(* CoDeSys 2.3 export: GVL_SYMBOLSANDDATATYPES.EXP *)

(* Global variable list: AdsClientTests/GVL_SymbolsAndDataTypes *)
VAR_GLOBAL PERSISTENT
	TestSymbol : STRING(82) := 'Some test value';(*Test comment äääöö*)
	TestDataType : ST_TestDataType;
END_VAR
